TYPE TcoControledZone_Info :
STRUCT
	{attribute addProperty Name "<#All#> - <#In automatic#>"}
	AllInAuto            : BOOL;
	
	{attribute addProperty Name "<#All#> - <#Is grounding#>"}
	AllInGrounding       : BOOL;
	
	{attribute addProperty Name "<#All#> - <#In manual#>"}
	AllInManual          : BOOL;
	
	{attribute addProperty Name "<#All#> - <#Idle#>"}
	AllIdle          : BOOL;

	{attribute addProperty Name "<#All#> - <#Grounded#>"}
	AllGrounded          : BOOL;
	
	{attribute addProperty Name "<#All#> - <#In step mode#>"}
	AllInStepMode        : BOOL;
	
	{attribute addProperty Name "<#All#> - <#Recovered#>"}
	AllRecovered        : BOOL;
	
	{attribute addProperty Name "<#All#> - <#Suspended#>"}
	AllSuspended        : BOOL;
	
	{attribute addProperty Name "<#All#> - <#Holding process#>"}
	AllHolding           : BOOL;
	
	{attribute addProperty Name "<#All#> - <#In Inactive or Manual or Grounded#>"}
	AllInactiveOrManualOrGrounded  : BOOL;
	
	{attribute addProperty Name "<#Group#> - <#Any station in automatic mode#>"}
	AnyInAuto            : BOOL;
	
	{attribute addProperty Name "<#Group#> - <#Any station in manual mode#>"}
	AnyInManual          : BOOL;
	
	{attribute addProperty Name "<#Group#> - <#Any station in step mode#>"}
	AnyInStepMode        : BOOL;
	
	{attribute addProperty Name "<#Group#> - <#Any station is grounding#>"}
	AnyGrounding         : BOOL;
	
	{attribute addProperty Name "<#Group#> - <#Any station is holded#>"}
	AnyInHolding         : BOOL;
	
	{attribute addProperty Name "<#Control panel#> - <#All keys in automatic#>"}
	AllKeysAuto          : BOOL;
	
	{attribute addProperty Name "<#Control panel#> - <#All keys in normal#>"}
	AllKeysNormal        : BOOL;
	
	{attribute addProperty Name "<#Control panel#> - <#Any key in manual#>"}
	AnyKeyManual         : BOOL;
	
	{attribute addProperty Name "<#Control panel#> - <#Any key in step#>"}
	AnyKeyStep           : BOOL;
	
	{attribute addProperty Name "<#Control panel#> - <#Any key in service#>"}
	AnyKeyService        : BOOL;
	
	{attribute addProperty Name "<#Control panel#> - <#Any button#> - <#Recover#>"}
	AnyButtonRecover       : BOOL;
	
	{attribute addProperty Name "<#Control panel#> - <#Any button#> - <#Suspend#>"}
	AnyButtonSuspend        : BOOL;
	
	{attribute addProperty Name "<#Control panel#> - <#Any button#> - <#Ground#>"}
	AnyButtonGround      : BOOL;
	
	{attribute addProperty Name "<#Control panel#> - <#Any button#> - <#Auto#>"}
	AnyButtonAuto     : BOOL;
	
	{attribute addProperty Name "<#Deadman#> - <#Any present#>"}
	AnyDeadmanPresent    : BOOL;

END_STRUCT
END_TYPE

(* stored: Version 1.1.0.1
   DUT TcoControledZone_Info: Id {aa141ebf-52fb-44f0-a6cb-185795382c0f} *)
